# EPICS substitutions: ioc/PhaseCavityTiming/PhaseCavityTimingApp/Db/IP231.substitutions
#==============================================================================
#
# Abs:  Acromag Analog Output IP-231 DAC template
#
# Name: IP231.substitutions
#
#  Auth: 10-Aug-2006, S. Peng         (PENG)
#  Rev:  dd-mmm-yyyy, Reviewer's Name (USERNAME)
#-----------------------------------------------------------------------------
# Mod:
#       dd-mmm-yyyy, First lastname (USERNAME):
#         comment
#
#==============================================================================
#
# EGU	- Engineering Units
# EGUF	- Engineering Units Full
# EGUL	- Engineering Units Low
# ADEL	- Archive Deadband Limit
# MDEL	- Monitor Deadband Limit
# HIHI	- HiHi Alarm Limit
# HIGH	- High Alarm Limit
# LOW	- Low  Alarm Limit
# LOLO	- LoLo Alarm Limit
#
file IP231.template
{
  pattern { RECORDNAME,           CH, EGUF,  EGUL,  ADEL,  MDEL, HIHI,  HIGH, LOW, LOLO, EGU   }
          { "$(CARD):out$(CH)",	0, 10.0,  -10.0, 0.0 ,  0.0 , 4.5 ,  4.0 , 1.0, 0.5,  Volts }
          { "$(CARD):out$(CH)",	1, 10.0,  -10.0, 0.0 ,  0.0 , 4.5 ,  4.0 , 1.0, 0.5,  Volts }
          { "$(CARD):out$(CH)",	2, 10.0,  -10.0, 0.0 ,  0.0 , 4.5 ,  4.0 , 1.0, 0.5,  Volts }
          { "$(CARD):out$(CH)",	3, 10.0,  -10.0, 0.0 ,  0.0 , 4.5 ,  4.0 , 1.0, 0.5,  Volts }
          { "$(CARD):out$(CH)",	4, 10.0,  -10.0, 0.0 ,  0.0 , 4.5 ,  4.0 , 1.0, 0.5,  Volts }
          { "$(CARD):out$(CH)",	5, 10.0,  -10.0, 0.0 ,  0.0 , 4.5 ,  4.0 , 1.0, 0.5,  Volts }
          { "$(CARD):out$(CH)",	6, 10.0,  -10.0, 0.0 ,  0.0 , 4.5 ,  4.0 , 1.0, 0.5,  Volts }
          { "$(CARD):out$(CH)",	7, 10.0,  -10.0, 0.0 ,  0.0 , 4.5 ,  4.0 , 1.0, 0.5,  Volts }
          { "$(CARD):out$(CH)",	8, 10.0,  -10.0, 0.0 ,  0.0 , 4.5 ,  4.0 , 1.0, 0.5,  Volts }
          { "$(CARD):out$(CH)",	9, 10.0,  -10.0, 0.0 ,  0.0 , 4.5 ,  4.0 , 1.0, 0.5,  Volts }
          { "$(CARD):out$(CH)", 10, 10.0,  -10.0, 0.0 ,  0.0 , 4.5 ,  4.0 , 1.0, 0.5,  Volts }
          { "$(CARD):out$(CH)", 11, 10.0,  -10.0, 0.0 ,  0.0 , 4.5 ,  4.0 , 1.0, 0.5,  Volts }
          { "$(CARD):out$(CH)", 12, 10.0,  -10.0, 0.0 ,  0.0 , 4.5 ,  4.0 , 1.0, 0.5,  Volts }
          { "$(CARD):out$(CH)", 13, 10.0,  -10.0, 0.0 ,  0.0 , 4.5 ,  4.0 , 1.0, 0.5,  Volts }
          { "$(CARD):out$(CH)", 14, 10.0,  -10.0, 0.0 ,  0.0 , 4.5 ,  4.0 , 1.0, 0.5,  Volts }
          { "$(CARD):out$(CH)", 15, 10.0,  -10.0, 0.0 ,  0.0 , 4.5 ,  4.0 , 1.0, 0.5,  Volts }
}
